FUNCTION_BLOCK FB_TankController IMPLEMENTS I_TankController
VAR_IN_OUT
	stTank : ST_Tank;
END_VAR
VAR
END_VAR


IF __ISVALIDREF(stTank) THEN
	CheckSafety();
	IF (stTank.bTemperatureAlarm) OR (stTank.bLevelAlarm) THEN
		IF stTank.bTemperatureAlarm THEN
			ApplyCooling();
			RETURN;
		END_IF
		IF stTank.bLevelAlarm THEN
			DispenseChemical();
		END_IF
	END_IF
	IF NOT (stTank.bTemperatureAlarm) AND NOT (stTank.bLevelAlarm) THEN
		TankProcessing();
	END_IF
END_IF

{warning 'add method implementation '}
METHOD ApplyCooling : BOOL

F_CoolTank(stTank);
END_METHOD

{warning 'add method implementation '}
METHOD CheckSafety : BOOL
F_CheckAlarm( pTank := ADR(stTank) )
END_METHOD

METHOD DispenseChemical : BOOL
VAR_INPUT
END_VAR
IF stTank.bLevelAlarm THEN
	TransferChemical( pTank := ADR(stTank) );
END_IF
END_METHOD

METHOD TankProcessing : BOOL
VAR_INPUT
END_VAR
stTank.fTemperature := stTank.fTemperature + GVL.fProcessTemperature;
stTank.fLevel := stTank.fLevel + GVL.fProcessLevel;
END_METHOD

END_FUNCTION_BLOCK

(* stored: Version 1.1.0.1, ProductVersion 3.1.4024.16
   POU FB_TankController: Id {d49f714c-8435-4f33-bc16-d19cf7467e69}, SpecialFunc None
   Method ApplyCooling: Id {c1b48702-0de2-4894-9461-4ad1944baf13}
   Method CheckSafety: Id {690d4314-9b02-4429-8769-3b48f9dada31}
   Method DispenseChemical: Id {d241761c-e1e3-4d70-816b-b992e91f2d02}
   Method TankProcessing: Id {39ed6fc7-899f-4f6a-9dac-2b7e80d90cff} *)
